# EPICS substitutions: elioApp/Db/EL1808.substitutions
file EL1808.template { pattern
{ CHAN	}
{ 1	}
{ 2	}
{ 3	}
{ 4	}
{ 5	}
{ 6	}
{ 7	}
{ 8	}
}
